Universal Robots PolyScope program: KI_Projekt_Roboterspiel_ET2_2022.urp

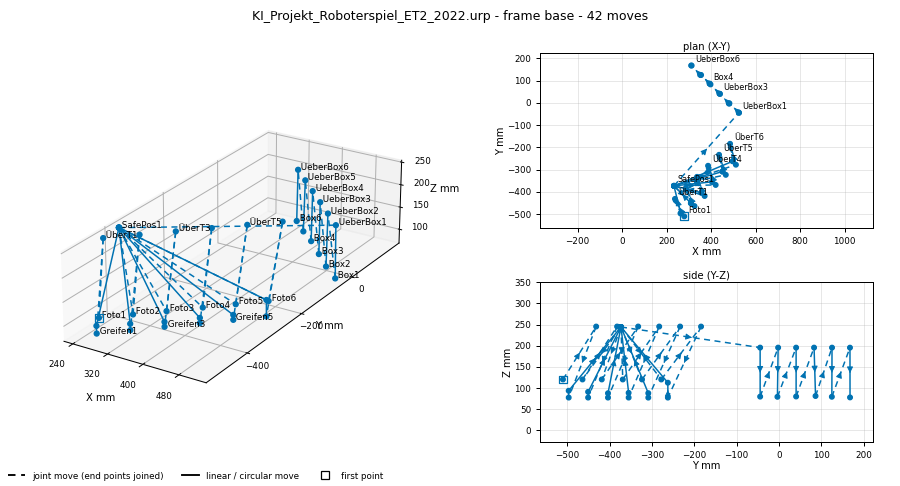
[picture p0: tool path of KI_Projekt_Roboterspiel_ET2_2022.urp in frame base, 42 of 42 moves have a stored position in this frame; points joined in program order, loops and branches not executed]
Program KI_Projekt_Roboterspiel_ET2_2022 (installation=default directory=/programs createdIn=3.8.0.61336 lastSavedIn=3.15.6.106324 robotSerialNumber=2019330179)
Calibrated DH parameters: a=[0.000106, -0.111627, -0.159498, 0.000094, -0.000086, 0]; d=[0.15209, -57.341072, 125.200339, -67.746952, 0.085336, 0.082359]; alpha=[1.571561, -0.003772, -0.00209, 1.571991, -1.571135, 0]; deltaTheta=[0.000042, 1.094313, -1.82127, 0.726912, -0.000025, -0.000055]
Robot Program (runOnlyOnce=true)
  Schrittnummer := 1
  Set ExpressionOutput pin=GP_int_out[0]; expression=0
  Wait Condition expression=GP_int_in[0]≟0
  x := 1
  Loop Counting (count=12) loopVariable(name=Schleife_1)
    Switch expression=Schrittnummer
      Case (caseValue=1)
        Switch expression=x
          Case (caseValue=1)
            MoveJ speed 60 deg/s, acceleration 80 deg/s^2 (useActiveTCP=true)
              Waypoint Foto1: TCP in base x=279.413 y=-510.25 z=120.423 mm, rx=-0.8077 ry=1.9846 rz=-1.6247 rad; joints [-266.905, -26.817, 83.486, -221.064, -51.024, 348.512] deg; flange x=185.971 y=-410.066 z=149.261 mm, rx=-0.8077 ry=1.9846 rz=-1.6247 rad
              Set ExpressionOutput pin=GP_int_out[0]; expression=1
              Wait Condition expression=GP_int_in[0]≠0
            MoveJ speed 60 deg/s, acceleration 80 deg/s^2 (useActiveTCP=true)
              Waypoint ÜberT1: TCP in base x=237.675 y=-431.845 z=245.374 mm, rx=-1.0775 ry=2.6966 rz=-0.9036 rad; joints [-259.969, -74.932, 76.748, -124.954, -78.224, 329.969] deg; flange x=195.833 y=-363.232 z=360.011 mm, rx=-1.0775 ry=2.6966 rz=-0.9036 rad
              URCap Greifer aktivieren (Robotiq_Grippers, Robotiq Inc.) dataModel(ResetAndActivateKey=false)
              URCap Greifer (Robotiq_Grippers, Robotiq Inc.) dataModel(position=50.0, force=100.0, speed=100.0, positionInDouble=50.0, forceInDouble=100.0, speedInDouble=100.0, slaveIds=[9], blocking=true)
              Waypoint Greifen1: TCP in base x=263.244 y=-496.719 z=77.616 mm, rx=-1.1687 ry=2.7832 rz=-0.3278 rad; joints [-256.757, -33.139, 35.464, -103.607, -82.267, 328.334] deg; flange x=238.161 y=-474.749 z=213.588 mm, rx=-1.1687 ry=2.7832 rz=-0.3278 rad
            URCap Greifer aktivieren (Robotiq_Grippers, Robotiq Inc.) dataModel(ResetAndActivateKey=false)
            URCap Greifer (Robotiq_Grippers, Robotiq Inc.) dataModel(position=90.58823529411765, force=48.0, speed=28.0, positionInDouble=90.58823529411765, forceInDouble=48.0, speedInDouble=28.0, slaveIds=[9], blocking=true)
            MoveL speed 250 mm/s, acceleration 1200 mm/s^2 (useActiveTCP=true) feature=Base
              Waypoint Anheben1: TCP in base x=263.212 y=-496.731 z=93.811 mm, rx=-1.1688 ry=2.7832 rz=-0.3278 rad; joints [-256.756, -33.15, 31.136, -99.27, -82.267, 328.342] deg; flange x=238.139 y=-474.755 z=229.783 mm, rx=-1.1688 ry=2.7832 rz=-0.3278 rad
              Waypoint SafePos1: TCP in base x=233.146 y=-373.178 z=244.335 mm, rx=-1.1705 ry=2.8033 rz=-0.2569 rad; joints [-256.319, -65.621, 44.927, -78.074, -83.498, 328.894] deg; flange x=212.17 y=-356.519 z=381.749 mm, rx=-1.1705 ry=2.8033 rz=-0.2569 rad
          Case (caseValue=2)
            MoveJ speed 60 deg/s, acceleration 80 deg/s^2 (useActiveTCP=true)
              Waypoint Foto2: TCP in base x=325.503 y=-464.154 z=120.417 mm, rx=-0.8076 ry=1.9848 rz=-1.6247 rad; joints [-258.363, -29.228, 90.951, -227.687, -59.29, 351.171] deg; flange x=232.075 y=-363.957 z=149.258 mm, rx=-0.8076 ry=1.9848 rz=-1.6247 rad
              Set ExpressionOutput pin=GP_int_out[0]; expression=1
              Wait Condition expression=GP_int_in[0]≠0
            MoveJ speed 60 deg/s, acceleration 80 deg/s^2 (useActiveTCP=true)
              Waypoint ÜberT2: TCP in base x=287.2 y=-382.332 z=245.411 mm, rx=-1.0776 ry=2.6965 rz=-0.9039 rad; joints [-249.739, -78.202, 81.343, -127.677, -83.934, 338.57] deg; flange x=245.354 y=-313.705 z=360.038 mm, rx=-1.0776 ry=2.6965 rz=-0.9039 rad
              URCap Greifer aktivieren (Robotiq_Grippers, Robotiq Inc.) dataModel(ResetAndActivateKey=false)
              URCap Greifer (Robotiq_Grippers, Robotiq Inc.) dataModel(position=50.0, force=100.0, speed=100.0, positionInDouble=50.0, forceInDouble=100.0, speedInDouble=100.0, slaveIds=[9], blocking=true)
              Waypoint Greifen2: TCP in base x=309.143 y=-450.819 z=77.622 mm, rx=-1.1689 ry=2.7832 rz=-0.3277 rad; joints [-250.121, -39.356, 47.758, -110.515, -83.636, 334.884] deg; flange x=284.07 y=-428.855 z=213.595 mm, rx=-1.1689 ry=2.7832 rz=-0.3277 rad
            URCap Greifer aktivieren (Robotiq_Grippers, Robotiq Inc.) dataModel(ResetAndActivateKey=false)
            URCap Greifer (Robotiq_Grippers, Robotiq Inc.) dataModel(position=90.58823529411765, force=48.0, speed=28.0, positionInDouble=90.58823529411765, forceInDouble=48.0, speedInDouble=28.0, slaveIds=[9], blocking=true)
            MoveL speed 250 mm/s, acceleration 1200 mm/s^2 (useActiveTCP=true) feature=Base
              Waypoint Anheben2: TCP in base x=309.132 y=-450.835 z=91.156 mm, rx=-1.1689 ry=2.7832 rz=-0.3277 rad; joints [-250.12, -39.867, 45.058, -107.304, -83.637, 334.893] deg; flange x=284.064 y=-428.873 z=227.131 mm, rx=-1.1689 ry=2.7832 rz=-0.3277 rad
              Waypoint SafePos2: TCP in base x=233.146 y=-373.178 z=244.335 mm, rx=-1.1705 ry=2.8033 rz=-0.2569 rad; joints [-256.319, -65.621, 44.927, -78.074, -83.498, 328.894] deg; flange x=212.17 y=-356.519 z=381.749 mm, rx=-1.1705 ry=2.8033 rz=-0.2569 rad
          Case (caseValue=3)
            MoveJ speed 60 deg/s, acceleration 80 deg/s^2 (useActiveTCP=true)
              Waypoint Foto3: TCP in base x=371.051 y=-418.604 z=120.434 mm, rx=-0.8077 ry=1.9846 rz=-1.6248 rad; joints [-248.49, -30.189, 94.241, -231.192, -68.887, 353.714] deg; flange x=277.612 y=-318.414 z=149.265 mm, rx=-0.8077 ry=1.9846 rz=-1.6248 rad
              Set ExpressionOutput pin=GP_int_out[0]; expression=1
              Wait Condition expression=GP_int_in[0]≠0
            MoveJ speed 60 deg/s, acceleration 80 deg/s^2 (useActiveTCP=true)
              Waypoint ÜberT3: TCP in base x=336.879 y=-332.615 z=245.431 mm, rx=-1.0776 ry=2.6966 rz=-0.9039 rad; joints [-238.271, -78.199, 81.503, -128.361, -90.497, 347.995] deg; flange x=295.043 y=-263.98 z=360.056 mm, rx=-1.0776 ry=2.6966 rz=-0.9039 rad
              URCap Greifer aktivieren (Robotiq_Grippers, Robotiq Inc.) dataModel(ResetAndActivateKey=false)
              URCap Greifer (Robotiq_Grippers, Robotiq Inc.) dataModel(position=50.0, force=100.0, speed=100.0, positionInDouble=50.0, forceInDouble=100.0, speedInDouble=100.0, slaveIds=[9], blocking=true)
              Waypoint Greifen3: TCP in base x=356.052 y=-403.908 z=77.592 mm, rx=-1.1686 ry=2.7833 rz=-0.3278 rad; joints [-242.719, -42.175, 53.354, -114.036, -85.244, 342.158] deg; flange x=330.973 y=-381.936 z=213.564 mm, rx=-1.1686 ry=2.7833 rz=-0.3278 rad
            URCap Greifer aktivieren (Robotiq_Grippers, Robotiq Inc.) dataModel(ResetAndActivateKey=false)
            URCap Greifer (Robotiq_Grippers, Robotiq Inc.) dataModel(position=90.58823529411765, force=48.0, speed=28.0, positionInDouble=90.58823529411765, forceInDouble=48.0, speedInDouble=28.0, slaveIds=[9], blocking=true)
            MoveL speed 250 mm/s, acceleration 1200 mm/s^2 (useActiveTCP=true) feature=Base
              Waypoint Anheben3: TCP in base x=356.014 y=-403.921 z=87.888 mm, rx=-1.1688 ry=2.7833 rz=-0.3278 rad; joints [-242.72, -42.705, 51.528, -111.681, -85.25, 342.158] deg; flange x=330.949 y=-381.942 z=223.861 mm, rx=-1.1688 ry=2.7833 rz=-0.3278 rad
              Waypoint SafePos3: TCP in base x=233.146 y=-373.178 z=244.335 mm, rx=-1.1705 ry=2.8033 rz=-0.2569 rad; joints [-256.319, -65.621, 44.927, -78.074, -83.498, 328.894] deg; flange x=212.17 y=-356.519 z=381.749 mm, rx=-1.1705 ry=2.8033 rz=-0.2569 rad
          Case (caseValue=4)
            MoveJ speed 60 deg/s, acceleration 80 deg/s^2 (useActiveTCP=true)
              Waypoint Foto4: TCP in base x=420.641 y=-369.009 z=120.396 mm, rx=-0.8076 ry=1.9847 rz=-1.6246 rad; joints [-236.644, -29.816, 93.191, -231.279, -80.458, 356.367] deg; flange x=327.206 y=-268.82 z=149.241 mm, rx=-0.8076 ry=1.9847 rz=-1.6246 rad
              Set ExpressionOutput pin=GP_int_out[0]; expression=1
              Wait Condition expression=GP_int_in[0]≠0
            MoveJ speed 60 deg/s, acceleration 80 deg/s^2 (useActiveTCP=true)
              Waypoint ÜberT4: TCP in base x=386.567 y=-282.924 z=245.397 mm, rx=-1.0774 ry=2.6968 rz=-0.9037 rad; joints [-226.476, -74.942, 77.186, -126.695, -97.231, 357.701] deg; flange x=344.75 y=-214.301 z=360.037 mm, rx=-1.0774 ry=2.6968 rz=-0.9037 rad
              URCap Greifer aktivieren (Robotiq_Grippers, Robotiq Inc.) dataModel(ResetAndActivateKey=false)
              URCap Greifer (Robotiq_Grippers, Robotiq Inc.) dataModel(position=50.0, force=100.0, speed=100.0, positionInDouble=50.0, forceInDouble=100.0, speedInDouble=100.0, slaveIds=[9], blocking=true)
              Waypoint Greifen4: TCP in base x=404.821 y=-355.158 z=77.657 mm, rx=-1.1688 ry=2.7832 rz=-0.328 rad; joints [-234.589, -42.198, 53.61, -114.848, -87.097, 350.084] deg; flange x=379.735 y=-333.166 z=213.624 mm, rx=-1.1688 ry=2.7832 rz=-0.328 rad
            URCap Greifer aktivieren (Robotiq_Grippers, Robotiq Inc.) dataModel(ResetAndActivateKey=false)
            URCap Greifer (Robotiq_Grippers, Robotiq Inc.) dataModel(position=90.58823529411765, force=48.0, speed=28.0, positionInDouble=90.58823529411765, forceInDouble=48.0, speedInDouble=28.0, slaveIds=[9], blocking=true)
            MoveL speed 250 mm/s, acceleration 1200 mm/s^2 (useActiveTCP=true) feature=Base
              Waypoint Anheben4: TCP in base x=404.814 y=-355.159 z=88.81 mm, rx=-1.1688 ry=2.7832 rz=-0.3281 rad; joints [-234.588, -42.777, 51.642, -112.302, -87.097, 350.092] deg; flange x=379.729 y=-333.164 z=224.776 mm, rx=-1.1688 ry=2.7832 rz=-0.3281 rad
              Waypoint SafePos4: TCP in base x=233.146 y=-373.178 z=244.335 mm, rx=-1.1705 ry=2.8033 rz=-0.2569 rad; joints [-256.319, -65.621, 44.927, -78.074, -83.498, 328.894] deg; flange x=212.17 y=-356.519 z=381.749 mm, rx=-1.1705 ry=2.8033 rz=-0.2569 rad
          Case (caseValue=5)
            MoveJ speed 60 deg/s, acceleration 80 deg/s^2 (useActiveTCP=true)
              Waypoint Foto5: TCP in base x=466.119 y=-323.553 z=120.473 mm, rx=-0.8076 ry=1.9846 rz=-1.6248 rad; joints [-225.595, -28.118, 87.947, -227.969, -91.269, 358.663] deg; flange x=372.682 y=-223.36 z=149.296 mm, rx=-0.8076 ry=1.9846 rz=-1.6248 rad
              Set ExpressionOutput pin=GP_int_out[0]; expression=1
              Wait Condition expression=GP_int_in[0]≠0
            MoveJ speed 60 deg/s, acceleration 80 deg/s^2 (useActiveTCP=true)
              Waypoint ÜberT5: TCP in base x=435.939 y=-233.565 z=245.369 mm, rx=-1.0776 ry=2.6967 rz=-0.9037 rad; joints [-215.357, -68.664, 68.136, -122.296, -103.385, 367.081] deg; flange x=394.113 y=-164.948 z=360.009 mm, rx=-1.0776 ry=2.6967 rz=-0.9037 rad
              URCap Greifer aktivieren (Robotiq_Grippers, Robotiq Inc.) dataModel(ResetAndActivateKey=false)
              URCap Greifer (Robotiq_Grippers, Robotiq Inc.) dataModel(position=50.0, force=100.0, speed=100.0, positionInDouble=50.0, forceInDouble=100.0, speedInDouble=100.0, slaveIds=[9], blocking=true)
              Waypoint Greifen5: TCP in base x=451.207 y=-308.708 z=77.537 mm, rx=-1.1688 ry=2.7832 rz=-0.3276 rad; joints [-226.729, -39.496, 48.677, -112.902, -88.931, 357.726] deg; flange x=426.138 y=-286.755 z=213.514 mm, rx=-1.1688 ry=2.7832 rz=-0.3276 rad
            URCap Greifer aktivieren (Robotiq_Grippers, Robotiq Inc.) dataModel(ResetAndActivateKey=false)
            URCap Greifer (Robotiq_Grippers, Robotiq Inc.) dataModel(position=90.58823529411765, force=48.0, speed=28.0, positionInDouble=90.58823529411765, forceInDouble=48.0, speedInDouble=28.0, slaveIds=[9], blocking=true)
            MoveL speed 250 mm/s, acceleration 1200 mm/s^2 (useActiveTCP=true) feature=Base
              Waypoint Anheben5: TCP in base x=451.22 y=-308.742 z=88.032 mm, rx=-1.1688 ry=2.7832 rz=-0.328 rad; joints [-226.727, -39.959, 46.713, -110.491, -88.937, 357.735] deg; flange x=426.137 y=-286.753 z=224 mm, rx=-1.1688 ry=2.7832 rz=-0.328 rad
              Waypoint SafePos5: TCP in base x=233.146 y=-373.178 z=244.335 mm, rx=-1.1705 ry=2.8033 rz=-0.2569 rad; joints [-256.319, -65.621, 44.927, -78.074, -83.498, 328.894] deg; flange x=212.17 y=-356.519 z=381.749 mm, rx=-1.1705 ry=2.8033 rz=-0.2569 rad
          Case (caseValue=6)
            MoveJ speed 60 deg/s, acceleration 80 deg/s^2 (useActiveTCP=true)
              Waypoint Foto6: TCP in base x=511.596 y=-278.066 z=120.357 mm, rx=-0.8076 ry=1.9849 rz=-1.6247 rad; joints [-215.139, -24.818, 78.498, -221.62, -101.508, 360.844] deg; flange x=418.179 y=-177.862 z=149.211 mm, rx=-0.8076 ry=1.9849 rz=-1.6247 rad
              Set ExpressionOutput pin=GP_int_out[0]; expression=1
              Wait Condition expression=GP_int_in[0]≠0
            MoveJ speed 60 deg/s, acceleration 80 deg/s^2 (useActiveTCP=true)
              Waypoint ÜberT6: TCP in base x=485.373 y=-184.12 z=245.327 mm, rx=-1.0776 ry=2.6966 rz=-0.9034 rad; joints [-205.43, -59.089, 52.94, -114.303, -108.565, 375.853] deg; flange x=443.534 y=-115.527 z=359.977 mm, rx=-1.0776 ry=2.6966 rz=-0.9034 rad
              URCap Greifer aktivieren (Robotiq_Grippers, Robotiq Inc.) dataModel(ResetAndActivateKey=false)
              URCap Greifer (Robotiq_Grippers, Robotiq Inc.) dataModel(position=50.0, force=100.0, speed=100.0, positionInDouble=50.0, forceInDouble=100.0, speedInDouble=100.0, slaveIds=[9], blocking=true)
              Waypoint Greifen6: TCP in base x=497.462 y=-262.477 z=77.584 mm, rx=-1.169 ry=2.7831 rz=-0.3278 rad; joints [-219.061, -33.527, 37.209, -107.468, -90.741, 365.157] deg; flange x=472.387 y=-240.502 z=213.556 mm, rx=-1.169 ry=2.7831 rz=-0.3278 rad
            URCap Greifer aktivieren (Robotiq_Grippers, Robotiq Inc.) dataModel(ResetAndActivateKey=false)
            URCap Greifer (Robotiq_Grippers, Robotiq Inc.) dataModel(position=90.58823529411765, force=48.0, speed=28.0, positionInDouble=90.58823529411765, forceInDouble=48.0, speedInDouble=28.0, slaveIds=[9], blocking=true)
            MoveL speed 250 mm/s, acceleration 1200 mm/s^2 (useActiveTCP=true) feature=Base
              Waypoint Anheben6: TCP in base x=497.416 y=-262.54 z=112.767 mm, rx=-1.1687 ry=2.7834 rz=-0.3278 rad; joints [-219.06, -33.173, 27.049, -97.658, -90.735, 365.188] deg; flange x=472.356 y=-240.562 z=248.741 mm, rx=-1.1687 ry=2.7834 rz=-0.3278 rad
              Waypoint SafePos6: TCP in base x=233.146 y=-373.178 z=244.335 mm, rx=-1.1705 ry=2.8033 rz=-0.2569 rad; joints [-256.319, -65.621, 44.927, -78.074, -83.498, 328.894] deg; flange x=212.17 y=-356.519 z=381.749 mm, rx=-1.1705 ry=2.8033 rz=-0.2569 rad
        Schrittnummer := 2
        x := x+1
      Case (caseValue=2)
        Switch expression=GP_int_in[0]
          Case (caseValue=1)
            MoveJ speed 60 deg/s, acceleration 80 deg/s^2 (useActiveTCP=true)
              Waypoint UeberBox1: TCP in base x=524.877 y=-44.568 z=195.666 mm, rx=-1.1474 ry=2.7862 rz=-0.3501 rad; joints [-194.125, -35.954, 9.104, -76.107, -97.082, 390.232] deg; flange x=498.82 y=-20.689 z=331.131 mm, rx=-1.1474 ry=2.7862 rz=-0.3501 rad
            MoveL speed 250 mm/s, acceleration 1200 mm/s^2 (useActiveTCP=true) feature=Base
              Waypoint Box1: TCP in base x=525.686 y=-44.519 z=79.866 mm, rx=-1.1476 ry=2.7861 rz=-0.35 rad; joints [-194.143, -42.725, 54.013, -114.257, -97.135, 390.164] deg; flange x=499.615 y=-20.648 z=215.33 mm, rx=-1.1476 ry=2.7861 rz=-0.35 rad
              URCap Greifer (Robotiq_Grippers, Robotiq Inc.) dataModel(position=0.0, force=48.0, speed=28.0, positionInDouble=0.0, forceInDouble=48.0, speedInDouble=28.0, slaveIds=[9], blocking=true)
            Set ExpressionOutput pin=GP_int_out[0]; expression=0
          Case (caseValue=2)
            MoveJ speed 60 deg/s, acceleration 80 deg/s^2 (useActiveTCP=true)
              Waypoint UeberBox2: TCP in base x=482.336 y=-2.071 z=195.643 mm, rx=-1.1474 ry=2.7863 rz=-0.3501 rad; joints [-190.019, -56.389, 46.338, -92.381, -98.05, 394.317] deg; flange x=456.29 y=21.816 z=331.109 mm, rx=-1.1474 ry=2.7863 rz=-0.3501 rad
            MoveL speed 250 mm/s, acceleration 1200 mm/s^2 (useActiveTCP=true) feature=Base
              Waypoint Box2: TCP in base x=481.014 y=-3.748 z=79.464 mm, rx=-1.1723 ry=2.7721 rz=-0.335 rad; joints [-190.682, -54.282, 74.481, -122.729, -97.19, 392.598] deg; flange x=454.581 y=18.386 z=215.153 mm, rx=-1.1723 ry=2.7721 rz=-0.335 rad
              URCap Greifer (Robotiq_Grippers, Robotiq Inc.) dataModel(position=0.0, force=48.0, speed=28.0, positionInDouble=0.0, forceInDouble=48.0, speedInDouble=28.0, slaveIds=[9], blocking=true)
            Set ExpressionOutput pin=GP_int_out[0]; expression=0
          Case (caseValue=3)
            MoveJ speed 60 deg/s, acceleration 80 deg/s^2 (useActiveTCP=true)
              Waypoint UeberBox3: TCP in base x=439.871 y=40.402 z=195.61 mm, rx=-1.1476 ry=2.7864 rz=-0.3501 rad; joints [-184.931, -67.218, 62.762, -97.237, -99.129, 399.375] deg; flange x=413.842 y=64.291 z=331.079 mm, rx=-1.1476 ry=2.7864 rz=-0.3501 rad
            MoveL speed 250 mm/s, acceleration 1200 mm/s^2 (useActiveTCP=true) feature=Base
              Waypoint Box3: TCP in base x=438.671 y=40.422 z=80.178 mm, rx=-1.1476 ry=2.7859 rz=-0.3504 rad; joints [-184.965, -62.533, 87.636, -126.843, -99.138, 399.257] deg; flange x=412.571 y=64.312 z=215.633 mm, rx=-1.1476 ry=2.7859 rz=-0.3504 rad
              URCap Greifer (Robotiq_Grippers, Robotiq Inc.) dataModel(position=0.0, force=48.0, speed=28.0, positionInDouble=0.0, forceInDouble=48.0, speedInDouble=28.0, slaveIds=[9], blocking=true)
            Set ExpressionOutput pin=GP_int_out[0]; expression=0
          Case (caseValue=4)
            MoveJ speed 60 deg/s, acceleration 80 deg/s^2 (useActiveTCP=true)
              Waypoint UeberBox4: TCP in base x=397.439 y=82.811 z=195.645 mm, rx=-1.1476 ry=2.7863 rz=-0.3501 rad; joints [-178.678, -75.259, 73.343, -98.752, -100.344, 405.625] deg; flange x=371.399 y=106.701 z=331.112 mm, rx=-1.1476 ry=2.7863 rz=-0.3501 rad
            MoveL speed 250 mm/s, acceleration 1200 mm/s^2 (useActiveTCP=true) feature=Base
              Waypoint Box4: TCP in base x=393.549 y=86.263 z=81.352 mm, rx=-1.1389 ry=2.7719 rz=-0.4093 rad; joints [-176.92, -69.795, 99.011, -130.905, -102.658, 407.066] deg; flange x=364.349 y=114.717 z=215.284 mm, rx=-1.1389 ry=2.7719 rz=-0.4093 rad
              URCap Greifer (Robotiq_Grippers, Robotiq Inc.) dataModel(position=0.0, force=48.0, speed=28.0, positionInDouble=0.0, forceInDouble=48.0, speedInDouble=28.0, slaveIds=[9], blocking=true)
            Set ExpressionOutput pin=GP_int_out[0]; expression=0
          Case (caseValue=5)
            MoveJ speed 60 deg/s, acceleration 80 deg/s^2 (useActiveTCP=true)
              Waypoint UeberBox5: TCP in base x=355.025 y=125.208 z=195.58 mm, rx=-1.1475 ry=2.7865 rz=-0.35 rad; joints [-171.097, -81.037, 79.923, -98.123, -101.65, 413.26] deg; flange x=329.006 y=149.096 z=331.05 mm, rx=-1.1475 ry=2.7865 rz=-0.35 rad
            MoveL speed 250 mm/s, acceleration 1200 mm/s^2 (useActiveTCP=true) feature=Base
              Waypoint Box5: TCP in base x=352.158 y=124.8 z=79.519 mm, rx=-1.1399 ry=2.7735 rz=-0.3541 rad; joints [-171.097, -75.322, 105.983, -130.773, -101.687, 413.162] deg; flange x=324.135 y=148.409 z=214.639 mm, rx=-1.1399 ry=2.7735 rz=-0.3541 rad
              URCap Greifer (Robotiq_Grippers, Robotiq Inc.) dataModel(position=0.0, force=48.0, speed=28.0, positionInDouble=0.0, forceInDouble=48.0, speedInDouble=28.0, slaveIds=[9], blocking=true)
            Set ExpressionOutput pin=GP_int_out[0]; expression=0
          Case (caseValue=6)
            MoveJ speed 60 deg/s, acceleration 80 deg/s^2 (useActiveTCP=true)
              Waypoint UeberBox6: TCP in base x=312.577 y=167.605 z=195.534 mm, rx=-1.1475 ry=2.7867 rz=-0.35 rad; joints [-162.186, -84.444, 83.077, -95.97, -102.931, 422.302] deg; flange x=286.583 y=191.505 z=331.008 mm, rx=-1.1475 ry=2.7867 rz=-0.35 rad
            MoveL speed 250 mm/s, acceleration 1200 mm/s^2 (useActiveTCP=true) feature=Base
              Waypoint Box6: TCP in base x=310.556 y=167.754 z=77.995 mm, rx=-1.1436 ry=2.7797 rz=-0.3516 rad; joints [-162.026, -78.078, 108.892, -128.593, -103.034, 422.354] deg; flange x=283.497 y=191.445 z=213.297 mm, rx=-1.1436 ry=2.7797 rz=-0.3516 rad
              URCap Greifer (Robotiq_Grippers, Robotiq Inc.) dataModel(position=0.0, force=48.0, speed=28.0, positionInDouble=0.0, forceInDouble=48.0, speedInDouble=28.0, slaveIds=[9], blocking=true)
            Set ExpressionOutput pin=GP_int_out[0]; expression=0
        Schrittnummer := 1
        MoveL speed 250 mm/s, acceleration 1200 mm/s^2 (useActiveTCP=true) feature=Base
          MoveDirectionNode (selectedDirection=ZPlus)
            Until DISTANCE (allowActions=false deceleration=3 distanceNodeType=STOP) Distance=0.05; motionParameters(blendRadius=0)
  Set ExpressionOutput pin=GP_int_out[0]; expression=99
  Wait Sleep waitTime=0.5
  Set ExpressionOutput pin=GP_int_out[0]; expression=0
